FUNCTION_BLOCK FB_TemperatureControl
VAR_INPUT
    bEnable     : BOOL;
    fSetpoint   : REAL;
    fActualTemp : REAL;
END_VAR

VAR_OUTPUT
    fControlOutput : REAL;   // -100 ... +100
    fHeatingPower  : REAL;   // 0 ... 100
    bCoolingValve  : BOOL;

    fError         : REAL;
END_VAR

VAR
    // PID parameters
    fK             : REAL := 100.0;
    fTN            : REAL := 30.0;
    fTV            : REAL := 5.0;

    // Controller states
    fIntegral      : REAL := 0.0;
    fDerivative    : REAL := 0.0;
    fPreviousError : REAL := 0.0;

    // 10 ms PLC task
    fCycleTime     : REAL := 0.01;

    // Cooling PWM
    fCoolingDemand : REAL := 0.0;
    tPWMElapsed    : TIME := T#0MS;
    tPWMOnTime     : TIME := T#0MS;
END_VAR

IF bEnable THEN

    // Control error

    fError := fSetpoint - fActualTemp;

    // Integral term

    fIntegral := fIntegral + (fError * fCycleTime / fTN);

    // Limit integral to avoid excessive wind-up
    fIntegral := LIMIT(-1.0, fIntegral, 1.0);

    // Derivative term

    fDerivative := fTV *(fError - fPreviousError) / fCycleTime;

	 fPreviousError := fError;

    // PID output

    fControlOutput := fK *(fError + fIntegral + fDerivative);

    // Controller output limit
    fControlOutput := LIMIT(-100.0, fControlOutput, 100.0);


ELSE

    fControlOutput := 0.0;
    fIntegral := 0.0;
    fDerivative := 0.0;
    fPreviousError := 0.0;

END_IF;


// Heating

IF fControlOutput > 0.0 THEN

    fHeatingPower := fControlOutput;
    fCoolingDemand := 0.0;

ELSE

    fHeatingPower := 0.0;
    fCoolingDemand := ABS(fControlOutput);

END_IF;

// Cooling PWM Period = 2 seconds

IF bEnable AND (fCoolingDemand > 0.0) THEN

    tPWMElapsed := tPWMElapsed + T#10MS;

    // Restart PWM cycle every 2 seconds
    IF tPWMElapsed >= T#2S THEN
        tPWMElapsed := T#0MS;
    END_IF;


    // Convert percentage to ON duration
    tPWMOnTime :=
        REAL_TO_TIME(
            (fCoolingDemand / 100.0) * 2000.0
        );


    bCoolingValve :=
        tPWMElapsed < tPWMOnTime;

ELSE

    bCoolingValve := FALSE;
    tPWMElapsed := T#0MS;

END_IF;

END_FUNCTION_BLOCK

(* stored: Version 1.1.0.1, ProductVersion 3.1.4024.16
   POU FB_TemperatureControl: Id {8e76f3c4-51ed-46f1-b00f-7368516f523f}, SpecialFunc None *)
